FUNCTION_BLOCK T_CantChangeStateFromIdleToSuspend EXTENDS T_UnitTestBase
VAR
  em : EquipmentModule;
  cmdTriggered : BOOL;
  actual, expected : E_PMLUnitMode;
  scanCounter : INT;
  myTestState : (ARRANGE, ACT, ASSERT);
END_VAR

CASE myTestState OF
  ARRANGE:
    CycleModuleLogicToAllowChangesToFilterThrough();

    IF em.InitComplete THEN
      em.ChangeState(E_PMLCommand.ePMLCommand_Clear);
      CycleModuleLogicToAllowChangesToFilterThrough();
      em.ChangeState(E_PMLCommand.ePMLCommand_Reset);
      CycleModuleLogicToAllowChangesToFilterThrough();
      myTestState := ACT;
    END_IF

  ACT:
    em.ChangeState(E_PMLCommand.ePMLCommand_Hold);
    CycleModuleLogicToAllowChangesToFilterThrough();
    actual := em.CurrentState;
    myTestState := ASSERT;

  ASSERT:
    assertion.AssertEquals_UINT(TO_UINT(actual), TO_UINT(E_PMLState.ePMLState_Idle), 'actual := em.CurrentState;');
    TestFinished();
END_CASE

METHOD CycleModuleLogicToAllowChangesToFilterThrough : BOOL
VAR_INST
	i: INT;

END_VAR
//em.CyclicLogic();
//CycleModuleLogicToAllowChangesToFilterThrough := i >= 100;
//i := SEL(i >= 100, i + 1, 0);

FOR i := 0 TO 100 DO
  em.CyclicLogic();
END_FOR
END_METHOD

END_FUNCTION_BLOCK

(* stored: Version 1.1.0.1, ProductVersion 3.1.4024.12
   POU T_CantChangeStateFromIdleToSuspend: Id {3cb9b207-189c-4f39-86b0-dd1023fa6ad6}, SpecialFunc None
   Method CycleModuleLogicToAllowChangesToFilterThrough: Id {2af72423-d40f-459a-9df6-e2a8b194de35} *)
